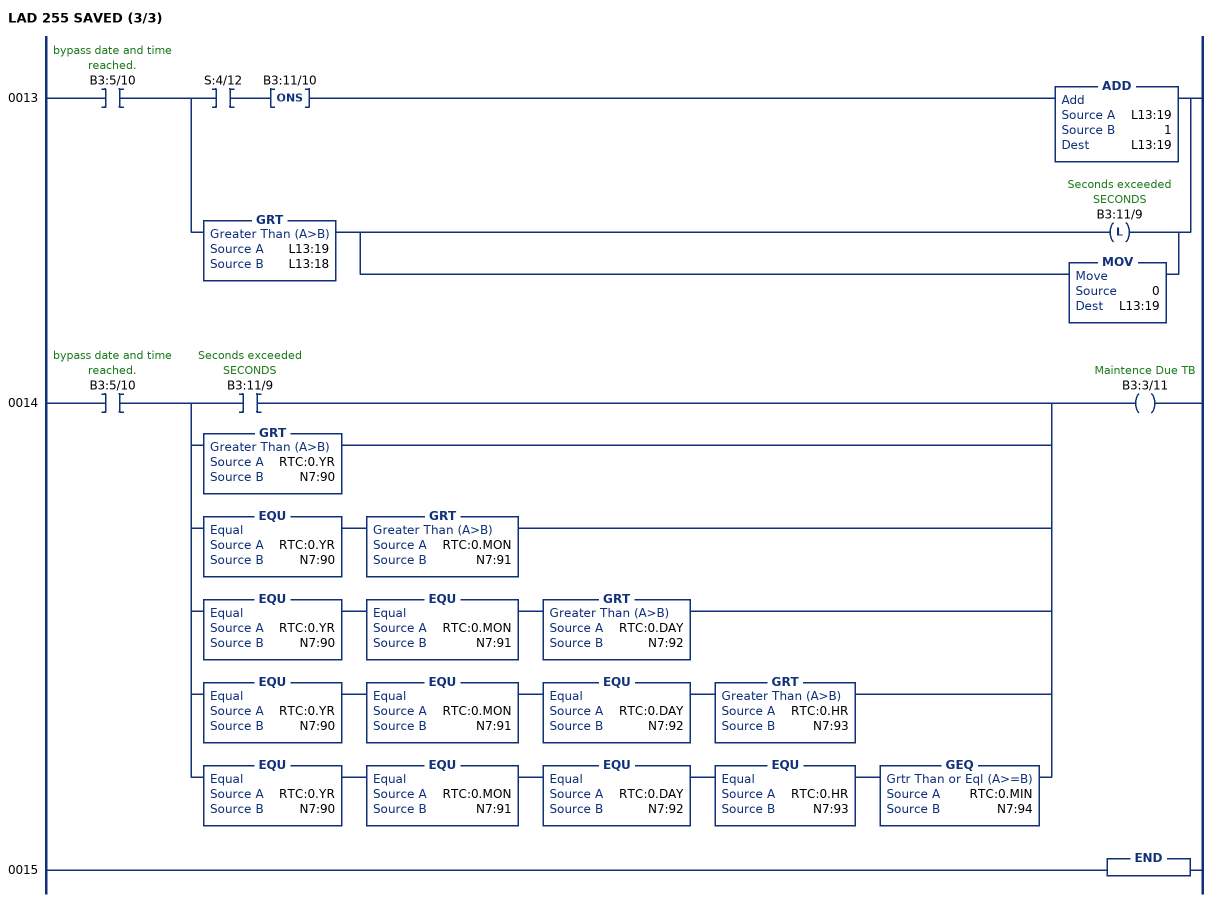
% Rung: 13 %
SOR XIC B3:5/10 BST XIC S:4/12 ONS B3:11/10 ADD L13:19 1 L13:19 NXB GRT L13:19 L13:18 BST OTL B3:11/9 NXB MOV 0 L13:19 BND BND EOR
%   B3:5/10  "bypass date and time reached." %
%   L13:18  MAX %
%   B3:11/9  SECONDS  "Seconds exceeded" %
% Rung: 14 %
SOR XIC B3:5/10 BST XIC B3:11/9 NXB GRT RTC:0.YR N7:90 NXB EQU RTC:0.YR N7:90 GRT RTC:0.MON N7:91 NXB EQU RTC:0.YR N7:90 EQU RTC:0.MON N7:91 GRT RTC:0.DAY N7:92 NXB EQU RTC:0.YR N7:90 EQU RTC:0.MON N7:91 EQU RTC:0.DAY N7:92 GRT RTC:0.HR N7:93 NXB EQU RTC:0.YR N7:90 EQU RTC:0.MON N7:91 EQU RTC:0.DAY N7:92 EQU RTC:0.HR N7:93 GEQ RTC:0.MIN N7:94 BND OTE B3:3/11 EOR
%   B3:5/10  "bypass date and time reached." %
%   B3:11/9  SECONDS  "Seconds exceeded" %
%   N7:90  RTC %
%   B3:3/11  TB  "Maintence Due" %
% Rung: 15 %
SOR END EOR

OTHER DOCUMENTED ADDRESSES
  B3:0/13  "toggle 2"
  B3:10/1  "bypass"
  B189:0/0  "change box"
  B189:0/9  "override boxing ok or not full signal"
  B189:0/11  "HMI force door close"
  B196:1/0  "Chute door is closed"
  B196:1/1  "control chute door"
  B196:1/13  "force box conveyor on"
  B196:3/0  "for hmi to continue production unlatched by hmi"
  HSC:0.0  "top"
  HSC:0.3/6  "Underflow interrupt"
  HSC:0.3/7  "Overflow interrupt"
  HSC:1.0  "bot"
  HSC:1.3/6  "Underflow interrupt"
  HSC:1.3/7  "Overflow interrupt"
  I:0.0/0  "Encoder Signal "A""
  I:0.0/1  "Encoder Signal "B""
  I:0.0/4  "Encoder Signal "A""
  I:0.0/5  "Encoder Signal "B""
  I:0.1/4  "not used"
  I:0.1/5  "not used"
  I:0.1/6  "not used"
  I:0.1/7  "not used"
  I:0.1/8  "not used"
  I:0.1/9  "not used"
  I:0.1/10  "not used"
  I:0.1/11  "not used"
  I:0.1/12  "not used"
  I:0.1/13  "not used"
  I:0.1/14  "not used"
  I:0.1/15  "not used"
  I:0.2  "not used"
  I:0.2/3  "Packaging Conveyor full"
  I:0.2/4  "Packaging Conveyor Box in Position"
  I:0.3  "not used"
  I:0.4  "Spare Analog Input 1"
  I:0.5  "Spare Analog Input 2"
  I:0.6  "Spare Analog Input 3"
  I:2.0/0  FRONT_ESTOP
  I:2.0/1  REAR_ESTOP
  I:2.0/8  FRONT_DOOR  "front door signal ce models only"
  I:2.0/9  REAR_DOOR  "rear door signal ce models only"
  I:2.0/11  "spare"
  L23:19  TOP_OPT_FAIL_CT
  L23:34  AIR_PRESSURE_FAULT
  L28:0  INS_1_TIME
  L29:0  INS_1_POS
  L30:0  INS_5_TIME
  L31:0  INS_5_POS
  L32:0  INS_6_TIME
  L33:0  INS_6_POS
  L192:1  BOT_LAST_TIME  "rtc bot belt previous movement event time"
  L192:2  BOT_CYCLE_TIME  "rtc bot belt time between events"
  L192:7  FROM_REAL  "distance from real part signal at optic location"
  L192:8  FROM_TRACKED  "distance from tracked part signal at optic location"
  L192:16  TOP_LAST_TIME  "rtc top belt previous movement event time"
  L192:17  TOP_CYCLE_TIME  "rtc top belt time between events"
  L199:5  ACQTM51
  L199:6  ACQTM52
  L199:7  ACQTM53
  L199:9  "ones"
  L199:10  "billions"
  L199:13  DUMP_LONG
  L199:15  ACQTM11
  L199:16  ACQTM12
  L199:17  ACQTM13
  L199:20  RESULTTM1
  L199:22  CLEARTIME5COUNT
  L199:23  CLEARTIME6COUNT
  L199:24  ACQTM61
  L199:25  ACQTM62
  L199:26  ACQTM63
  L199:27  TMSINCETRIG1
  L199:29  TMSINCETRIG5
  L199:30  TMSINCETRIG6
  L199:31  CLEARTIME1COUNT
  L199:32  RESULTTM5
  L199:33  RESULTTM6
  L199:34  MAXACQTM1
  L199:36  MAXACQTM6
  N7  
  N101:2  I3_TRIG_LOC
  N101:3  I4_TRIG_LOC
  O:0.0/1  "spare"
  O:0.0/11  "Spare"
  O:0.0/12  "not used"
  O:0.0/13  "not used"
  O:0.0/14  "not used"
  O:0.0/15  "not used"
  O:0.1  "not used"
  O:0.2  "not used"
  O:0.3  "not used"
  O:0.5  "spare analog output"
  O:3.0/0  "spare"
  O:3.0/2  "spare"
  O:3.0/3  "light curtain range selection /* needed? */"
  O:3.0/7  "door unlocks on CE models"
  O:3.0/8  "Light?"
  PFILE:6  "check for part jams"
  PFILE:10  "Bottom belt HSC"
  PFILE:12  "Top belt HSC"
  Q2:55  END_OF_MAIN
  Q5:94  END_OF_BELTS
  T20:0  "Trigger On Time"
  U:9  "slow data"
  U:24  "check skipped fail rate"
  U:28  "faults"
  U:29  "speed"
  U:30  "count"
  U:31  "rate calc"
  U:32  "boxer"
  U:33  "bulk pack"
  U:34  "customer boxing unit signals"
  U:35  "cleanup"

COMMENTS NOT ATTACHED TO A CURRENT RUNG
  R6:2: B41 is the top good 3 file
  R6:6/DN: B35 is the top NG file
  R6:10/DN: B37 is the top good 1 file
  R6:11/DN: B39 is the top good 2 file
  R6:0: B36 is the bottom GOOD file
  R6:10: B37 is the top good 1 file
  R6:6: B35 is the top NG file
  R6:4: B34 is the bottom NG file

REVISION NOTES
  13: updated count reset
  14: added io moduals
  15: multiple steps toward new hmi integration
  21: test
  27: fix error if bulk pack and no boxing fallout were on

DATA TABLE (non-zero values as saved)
DATA B3
% B3:0 % 0X8036 0X1360 0X4001 0XA501 0X0EFB 0X0570 0X15B8 0X0421 0X2F80 0X22D0
% B3:10 % 0X21FC 0X00CE 0X4000 0X8000 0X0000 0X0000 0X0000 0X0000 0X0000 0X0000
% B3:50 % 0X0001 0X0000 0X0000 0X0000 0X0000 0X0000 0X0000 0X0000 0X0000 0X0000
DATA T4
% .PRE .ACC %
% T4:0 % 0 1
% T4:1 % 150 0
% T4:2 % 400 0
% T4:3 % 250 127
% T4:4 % 1000 1000
% T4:5 % 5 5
% T4:6 % 10 10
% T4:7 % 150 0
% T4:8 % 20 0
% T4:9 % 50 17
% T4:10 % 200 200
% T4:11 % 111 0
% T4:12 % 20 20
% T4:13 % 250 0
% T4:14 % 666 0
% T4:15 % 1000 1001
% T4:16 % 400 0
% T4:17 % 100 14
% T4:18 % 5 0
% T4:19 % 300 0
% T4:20 % 200 0
% T4:21 % 200 0
% T4:22 % 200 0
% T4:23 % 250 0
% T4:24 % 666 0
% T4:25 % 666 0
% T4:26 % 666 0
% T4:27 % 250 0
% T4:28 % 250 0
% T4:29 % 5000 0
% T4:30 % 333 140
% T4:31 % 333 156
% T4:32 % 250 176
% T4:33 % 250 181
DATA C5
% .PRE .ACC %
% C5:0 % 32766 0
DATA R6
% .LEN .POS %
% R6:0 % 1250 0
% R6:1 % 16 0
% R6:2 % 1050 0
% R6:3 % 1050 0
% R6:4 % 1250 0
% R6:5 % 1250 0
% R6:6 % 1713 0
% R6:7 % 16 0
% R6:8 % 1024 0
% R6:9 % 3 0
% R6:10 % 1713 0
% R6:11 % 1050 0
% R6:12 % 10 0
% R6:13 % 10 0
% R6:14 % 10 0
% R6:15 % 10 0
% R6:16 % 1713 0
% R6:17 % 1713 0
% R6:18 % 1050 0
% R6:19 % 10 0
DATA N7
% N7:0 % 17248 4 1009 300 3 0 0 0 500 43
% N7:10 % 1000 43 0 2 20 20 1000 2000 50 1050
% N7:20 % 0 1329 10 2000 222 46 0 0 0 250
% N7:30 % 666 1420 150 0 0 1231 77 25 0 25
% N7:40 % 3 37 0 37 32767 482 1224 1350 1636 15
% N7:50 % 14 16 15 16 17 1024 0 0 32766 3
% N7:60 % 1713 1713 1050 984 1034 1024 4999 5 400 400
% N7:70 % 100 200 300 400 90 190 290 390 16835 15892
% N7:80 % 0 0 1249 1255 1300 1310 42 36 0 0
% N7:90 % 2011 4 4 12 1 42 36 222 222 12
% N7:100 % 1003 90 110 100 175 25 0 0 0 0
% N7:190 % -128 27477 27605 32767 0 0 0 0 0 0
DATA F8
% F8:0 % 6
DATA L13
% L13:0 % 12164 115616 0 36561 172395
% L13:5 % 1563 5514 1563 142278 1
% L13:10 % 1 13 30834 15 90
% L13:15 % -1579716633 -2147483648 2147483647 2147483647 82058
% L13:20 % 68189453 -2107658304 777 34576 100
% L13:25 % 121 2245 -27180 0 -1580393830
% L13:30 % 676781 1563 1020000 1572502331 444
% L13:35 % 0 36 99 -1248231873 -1248231801
% L13:40 % 25576 1000000000 1000000 1572502304 -1579813256
% L13:45 % -1579813239 72 0 27 20163346
% L13:50 % 96667 1842945 -1579914627 0 0
% L13:55 % 96650 23729 18356 0 -1783954972
% L13:60 % 26 104 -1783954986 600 6
% L13:65 % 100 600 -1248227341 -1248227308 12
% L13:70 % -2107767826 11 118 2557600 20163346
% L13:75 % 922236 60 100 -1579914616 2
% L13:80 % 24 74 148 7 1835572
% L13:85 % 55788 290 289 0 96711
% L13:90 % 96694 5 36308 5 -1579813231
% L13:95 % 10 256 0 -1579813214 89418
% L13:100 % 182972200 6 1600 14 505
% L13:105 % 89418 31 68131605 27211 68131598
% L13:110 % 7 100 50 -2107714067 -2107714068
% L13:115 % -2107714054 14 7 -2107714061 26
% L13:120 % 12 27206 50 100 10
% L13:125 % 0 -2107767826 -1050 3276500 55826
% L13:130 % 2 2 0 99 0
% L13:135 % 0 0 55813 5 70
% L13:140 % 0 5 36 50 50
% L13:145 % 1843080 5 5 5 19
% L13:150 % 12 20 27193 -27193 13
% L13:155 % 0 -10 0 0 4589052
% L13:160 % 15 25 25 1220 45
% L13:165 % -2107713833 -2107713823 -2107713833 -2107713823 6706
% L13:170 % 12817 47350 47349 800 200
% L13:175 % 4 4 42 23 38
% L13:180 % -1248213949 77 50757 1000000 289000000
% L13:185 % 0 1 -1248213836 77 50896
% L13:190 % 290000000 0 0 0 0
DATA L19
% L19:0 % -1580384158 -1580384071 -1580365159 -1580202793 -1580177296
% L19:5 % -1580161804 -1580144655 -1580115967 -1580083679 -1580061191
% L19:10 % -1579987131 -1579984507 -1579861709 -1579860988 -1579813640
% L19:15 % -1580393830 -1580384242 0 0 0
DATA L20
% L20:0 % -1580422411 -1580422157 -1580421901 -1580421646 -1580393447
% L20:5 % -1580383857 -1580383774 -1580383689 -1580364776 -1580202410
% L20:10 % -1580176912 -1580161420 -1580144271 -1580126885 -1580126627
% L20:15 % -1580125349 -1580125091 -1580124834 -1580115583 -1580094755
% L20:20 % -1580094500 -1580094244 -1580093987 -1580093732 -1580093476
% L20:25 % -1580093222 -1580092967 -1580092713 -1580083280 -1580060795
% L20:30 % -1579986736 -1579984109 -1579916608 -1579915090 -1579914583
% L20:35 % -1579882876 -1579882623 -1579881347 -1579881090 -1579880837
% L20:40 % -1579861324 -1579860606 -1579813256 -1580792699 -1580791181
% L20:45 % -1580680495 -1580423428 -1580423173 -1580422920 -1580422666
DATA L21
% L21:0 % -2108048522 -2108048439 -2108048359 -2108048283 -2108037091
% L21:5 % -2108031581 -2108031533 -2108031484 -2108020617 -2107927324
% L21:10 % -2107912674 -2107903772 -2107893920 -2107883931 -2107883783
% L21:15 % -2107883049 -2107882900 -2107882753 -2107877437 -2107865476
% L21:20 % -2107865341 -2107865213 -2107865090 -2107864975 -2107864866
% L21:25 % -2107864764 -2107864667 -2107864575 -2107861147 -2107848657
% L21:30 % -2107807594 -2107806138 -2107768754 -2107768034 -2107767806
% L21:35 % -2107753741 -2107753618 -2107752955 -2107752814 -2107752673
% L21:40 % -2107741452 -2107741039 -2107713833 -2108212679 -2108212006
% L21:45 % -2108162912 -2108048900 -2108048798 -2108048702 -2108048610
DATA L22
% L22:0 % -1580383757 -1580383672 -1580364759 -1580202392 -1580176895
% L22:5 % -1580161402 -1580144254 -1580126864 -1580126605 -1580125327
% L22:10 % -1580125071 -1580124815 -1580115566 -1580094736 -1580094480
% L22:15 % -1580094226 -1580093973 -1580093717 -1580093462 -1580093207
% L22:20 % -1580092952 -1580092698 -1580083262 -1580060777 -1579986718
% L22:25 % -1579984091 -1579916564 -1579915042 -1579914536 -1579882849
% L22:30 % -1579882594 -1579881313 -1579881058 -1579880802 -1579861307
% L22:35 % -1579860588 -1579813239 -1580791160 -1580790655 -1580680472
% L22:40 % -1580423410 -1580423156 -1580422902 -1580422648 -1580422394
% L22:45 % -1580422139 -1580421884 -1580421630 -1580393429 -1580383840
DATA L23
% L23:0 % -2108031523 -2108031474 -2108020607 -2107927314 -2107912664
% L23:5 % -2107903762 -2107893910 -2107883919 -2107883770 -2107883036
% L23:10 % -2107882889 -2107882742 -2107877427 -2107865466 -2107865331
% L23:15 % -2107865204 -2107865084 -2107864969 -2107864860 -2107864759
% L23:20 % -2107864662 -2107864570 -2107861137 -2107848647 -2107807584
% L23:25 % -2107806128 -2107768732 -2107768013 -2107767785 -2107753728
% L23:30 % -2107753604 -2107752937 -2107752796 -2107752653 -2107741442
% L23:35 % -2107741029 -2107713823 -2108211997 -2108211773 -2108162902
% L23:40 % -2108048892 -2108048792 -2108048695 -2108048604 -2108048516
% L23:45 % -2108048433 -2108048354 -2108048278 -2108037081 -2108031571
DATA L30
% L30:0 % 1097513510 1097513738 1097513967 1097514196 1097514426
% L30:5 % 1097514655 1097514883 1097515111 1097515339 1569237509
% L30:10 % 1571789345 1571789602 1571790886 1571791144 1571791400
% L30:15 % 1572418698 1572420630 1572420885 1572422166 1572422422
% L30:20 % 1572422681 1572500242 1572500500 1572501791 1572502048
% L30:25 % 1572502304 1071308573 1071308799 1071309024 1071309250
% L30:30 % 1071309476 1071429569 1071429795 1071431153 1071431379
% L30:35 % 1071431606 1088333039 1088333266 1088334623 1088334848
% L30:40 % 1088335075 1089808842 1089809070 1089810430 1089810657
% L30:45 % 1089810882 1092780028 1092791426 1092806921 1097513283
DATA L31
% L31:0 % 3522828 3522897 3522967 3523035 3523105
% L31:5 % 3523175 3523244 3523313 3523382 18677621
% L31:10 % 19955820 19955950 19956596 19956726 19956855
% L31:15 % 20121868 20122368 20122448 20122938 20123054
% L31:20 % 20123174 20162306 20162436 20163087 20163217
% L31:25 % 20163346 2077757 2077757 2077757 2077757
% L31:30 % 2077757 2077757 2077757 2077757 2077757
% L31:35 % 2077757 2077757 2077757 2077757 2077757
% L31:40 % 2077757 2077757 2077757 2077757 2077757
% L31:45 % 2077757 2091375 2094821 2099507 3522760
DATA L32
% L32:0 % -1580899456 -1580898953 -1580898345 -1580897704 -1580897358
% L32:5 % -1580896765 -1580896275 -1580895067 -1580894460 -1580894137
% L32:10 % -1580893486 -1580892228 -1580890645 -1580889936 -1580886285
% L32:15 % -1580885998 -1580885480 -1580884222 -1580883798 -1580882366
% L32:20 % -1580881379 -1580881061 -1580880684 -1580880188 -1580879250
% L32:25 % -1580878973 -1580878469 -1580877903 -1580872167 -1580792721
% L32:30 % -1580791202 -1580790695 -1580680535 -1579920498 -1579920134
% L32:35 % -1579916653 -1579915132 -1579914627 -1580906522 -1580906306
% L32:40 % -1580906076 -1580905803 -1580905334 -1580905154 -1580901792
% L32:45 % -1580901242 -1580900843 -1580900268 -1580900094 -1580899829
DATA L33
% L33:0 % -2108260033 -2108259810 -2108259540 -2108259256 -2108259102
% L33:5 % -2108258839 -2108258622 -2108258086 -2108257817 -2108257674
% L33:10 % -2108257385 -2108256827 -2108256125 -2108255810 -2108254191
% L33:15 % -2108254064 -2108253834 -2108253276 -2108253088 -2108252453
% L33:20 % -2108252015 -2108251874 -2108251707 -2108251487 -2108251071
% L33:25 % -2108250948 -2108250724 -2108250473 -2108247929 -2108212689
% L33:30 % -2108212015 -2108211791 -2108162930 -2107770872 -2107770670
% L33:35 % -2107768776 -2107768053 -2107767826 -2108263167 -2108263071
% L33:40 % -2108262969 -2108262848 -2108262640 -2108262560 -2108261069
% L33:45 % -2108260825 -2108260648 -2108260393 -2108260316 -2108260198
DATA B40
% B40:0 % 0XAAAA
DATA B41
% B41:60 % 0X0000 0X0000 0X0000 0X0002 0X0000 0X0000 0X0000 0X0000 0X0000 0X0000
DATA B100
% B100:0 % 0X2700 0X18A0 0X0004 0X0000 0X0000 0X0000 0X0000 0X0000 0X0000 0X0000
DATA N101
% N101:0 % 118 17365 0 0 1183 100 1002 1200 1212 1230
% N101:10 % 1240 1604 10 14089 1269 0 3297 250 333 333
% N101:20 % 1000 500 400 0 0 0 250 250 0 0
DATA L102
% L102:0 % 20 10 5687 5701 5700
% L102:5 % 5700 2 0 0 0
% L102:10 % 0 0 0 0 36308
% L102:15 % 0 30 10 30 10
% L102:20 % 0 8 69362 0 25
% L102:25 % 27 0 1829722 81649 714735
% L102:30 % 11 0 16 7754 3
% L102:35 % 0 302 0 999999 25
% L102:40 % 0 2 63160 0 0
